Staubli VAL3: aioItem.pjx

--- aioItem.pjx ---
Parameters version=s7.2.1 stackSize=5000 millimeterUnit=true
Data file=aioItem.dtx

--- aioItem.dtx ---
public bool bActive
public string sID
public string sName
public aio aAio
public bool bEnable
